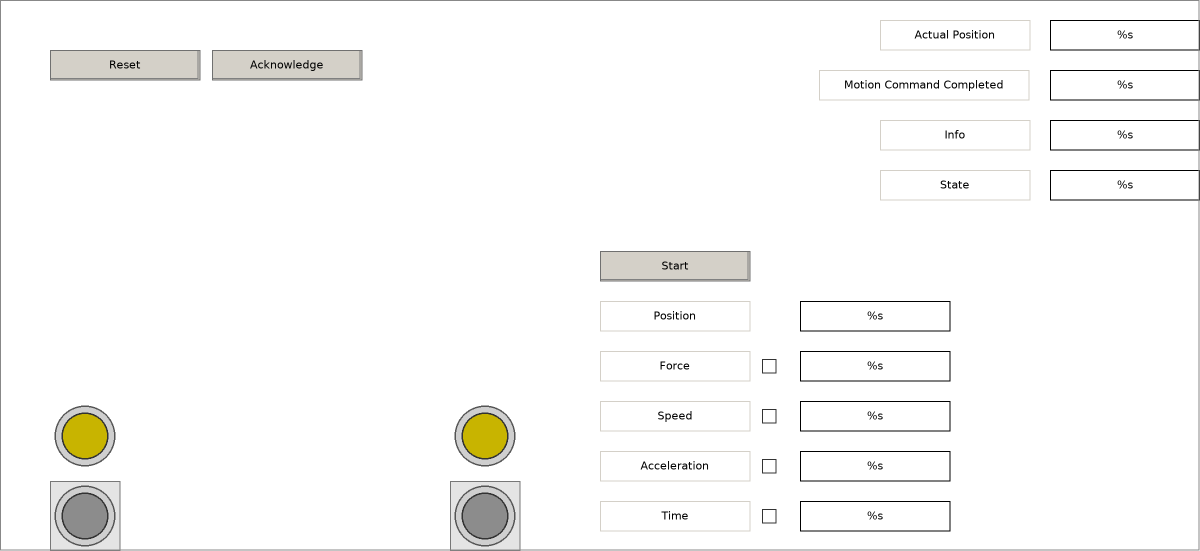
VISUALIZATION VisualizationTest  // 1200x551
    Checkbox (760,351 30x30), variable: MAIN.CylTronicCylinder1.ForceActive
    Checkbox (760,401 30x30), variable: MAIN.CylTronicCylinder1.SpeedActive
    Checkbox (760,451 30x30), variable: MAIN.CylTronicCylinder1.AccelerationActive
    Textfield (600,351 150x30), "Force"
    Textfield (600,401 150x30), "Speed"
    Textfield (600,451 150x30), "Acceleration"
    Textfield (600,301 150x30), "Position"
    Textfield (600,501 150x30), "Time"
    Checkbox (760,501 30x30), variable: MAIN.CylTronicCylinder1.TimeActive
    Rectangle (800,301 150x30), "%s", text variable: MAIN.CylTronicCylinder1.Pos
        OnMouseClick: write the text variable via VisuDialogs.Numpad, min MAIN.CylTronicCylinder1.MinPos, max MAIN.CylTronicCylinder1.MaxPos
    Rectangle (92,274 258x100)
    Rectangle (350,308 150x30)
    Lamp1 (50,401 70x70), variable: MAIN.CylTronicCylinder1.DataIn.CyltronicDataInAct.LimitSwitchOut, style: Lamp-Lamp1-Yellow
    Lamp1 (450,401 70x70), variable: MAIN.CylTronicCylinder1.DataIn.CyltronicDataInAct.LimitSwitchOut, style: Lamp-Lamp1-Yellow
    PushSwitch (50,481 70x70), variable: MAIN.CylTronicCylinder1.In, behaviour: TAP, style: Switch-PushSwitch-Gray
    PushSwitch (450,481 70x70), variable: MAIN.CylTronicCylinder1.Out, behaviour: TAP, style: Switch-PushSwitch-Gray
    Button (600,251 150x30), "Start"
        OnMouseClick: toggle MAIN.CylTronicCylinder1.Start
    Button (50,50 150x30), "Reset"
        OnMouseClick: toggle MAIN.CylTronicCylinder1.Reset
    Button (212,50 150x30), "Acknowledge"
        OnMouseClick: toggle MAIN.CylTronicCylinder1.Acknowledge
    Rectangle (800,351 150x30), "%s", text variable: MAIN.CylTronicCylinder1.Force
        OnMouseClick: write the text variable via VisuDialogs.Numpad, min 0, max 20
    Rectangle (800,401 150x30), "%s", text variable: MAIN.CylTronicCylinder1.Speed
        OnMouseClick: write the text variable via VisuDialogs.Numpad, min 0, max 600
    Rectangle (800,451 150x30), "%s", text variable: MAIN.CylTronicCylinder1.Acceleration
        OnMouseClick: write the text variable via VisuDialogs.Numpad, min 0, max 20
    Rectangle (800,501 150x30), "%s", text variable: MAIN.CylTronicCylinder1.Time0
        OnMouseClick: write the text variable via VisuDialogs.Numpad, min 0, max 20000
    Rectangle (1050,20 150x30), "%s", text variable: MAIN.CylTronicCylinder1.DataIn.CyltronicDataInAct.ActualPosition
    Textfield (880,20 150x30), "Actual Position"
    Rectangle (1050,70 150x30), "%s", text variable: MAIN.CylTronicCylinder1.DataIn.CyltronicDataInAct.MotionCommandCompleted
    Textfield (819,70 210x30), "Motion Command Completed"
    Rectangle (1050,120 150x30), "%s", text variable: MAIN.CylTronicCylinder1.Meldung
    Textfield (880,120 150x30), "Info"
    Rectangle (1050,170 150x30), "%s", text variable: MAIN.CylTronicCylinder1.StateText
    Textfield (880,170 150x30), "State"
END_VISUALIZATION

(* stored: Version 1.1.0.1, ProductVersion 3.1.4024.10
   Visu VisualizationTest: Id {2db9162b-44e7-4540-a78b-5eb1fdae9ec7} *)
